Staubli VAL3: BeforeArrayCut.pgx

public program BeforeArrayCut(num x_nWorkplaceIn, num x_nTrajindex)
begin
  //参数：x_nWorkplaceIn 工位序号，传入的参数是 DataBase:nWorkPlaceIndex
  //参数：x_nTrajIndex 路径序号，传入的参数是TxtFile:nReadTrajIndex
  //引用位置:Motion:Move.pgx
  //功能：在阵列之前添加动作
  //备注：添加动作需要waitendmove()
  //







end
